{attribute addProperty BoxType "EL5101-0011-0016"}
{attribute addProperty Id "ControlAT %Q*Control_879818281620Set_counter_valueAT %Q*UDINT32417"}
{attribute addProperty CRC "22981790"}
{attribute addProperty SizeInBites "48"}
{attribute addProperty SizeInBytes "6"}
TYPE ENC_Control_015EAC9E :
STRUCT
	{attribute addProperty Name "Control"}
	Control AT %Q* : Control_87981828;
	{attribute addProperty Name "Set_counter_value"}
	Set_counter_value AT %Q* : UDINT;
END_STRUCT
END_TYPE

(* stored: Version 1.2.0.0, ProductVersion 3.1.4024.9
   DUT ENC_Control_015EAC9E: Id {c34f3aaa-01d2-4d02-b5d4-eb76c67b321a} *)
